// TwinCAT 3 PLC project ZeroTorque
// ProgramVersion: 3.1.4020.4
// libraries:
//   Tc2_MC2, * (Beckhoff Automation GmbH)
//   Tc2_Standard, * (Beckhoff Automation GmbH)
//   Tc2_System, * (Beckhoff Automation GmbH)
//   Tc3_Module, * (Beckhoff Automation GmbH)
// project tree:
//   GVLs/ GVL.TcGVL
//   / PlcTask.TcTTO
//   POUs/ KalmanFilter.TcPOU, MAIN.TcPOU
// real-time tasks:
//   TASK PlcTask: cycle T#10ms, priority 20, ADS port 350
// motion (NC):
//   TASK NC-Task 1 SAF: cycle T#2ms, priority 4, ADS port 501
//   TASK NC-Task 1 SVB: cycle T#10ms, priority 8, ADS port 511
//   AXIS Axis 1 (id 1)
//     Dynamic: AccelerationMaximum=150000, DecelerationMaximum=150000, Acceleration=5566, Deceleration=5566, Jerk=5566
//     Velo: SlowManual=50000, FastManual=150000, Maximum=150000
//     PositionAreaControl: Enable=false, RefSearch=false
//     TargetPosControl: Enable=false
//     OtherSettings: AllowMotionCmdToSlave=true
//     encoder EncType=19
//       EncPara: ScaleFactorNumerator=1, MaxCount=#xffffffff
//     drive DrvType=16
//       DrvPara: MaxCount=#xffffffff
//         Analog: VeloReferenz=150000
//         TimeComp: TaskDelayCycles=1
//     controller CtrType=1
//       CtrPara: PriorControlFactor=1
//         PosDiffControl: Enable=false
//         Observer: BandWidth=20
// I/O:
//   DEVICE Device 3 (EtherCAT), AmsNetId 172.18.138.230.4.1
//     Drive 1 (ZeroErr Driver) [ZeroErr Driver]
// variable links:
//   NC-Task 1 SAF/Axes/Axis 1 <-> Device 3 (EtherCAT)/Drive 1 (ZeroErr Driver)
//     Drive/Inputs/In/nDcOutputTime <-> InfoData/DcOutputShift
//     Drive/Inputs/In/nState1 <-> Transmit PDO mapping 0/Status word
//     Drive/Inputs/In/nState2 <-> Transmit PDO mapping 0/Status word @bit 8
//     Drive/Inputs/In/nState4 @bit 1 <-> WcState/InputToggle
//     Drive/Inputs/In/nState4 <-> WcState/WcState
//     Drive/Outputs/Out/nCtrl1 <-> Receive PDO mapping 0/Control word
//     Drive/Outputs/Out/nCtrl2 <-> Receive PDO mapping 0/Control word @bit 8
//     Drive/Outputs/Out/nDataOut1 <-> Receive PDO mapping 0/Target Position
//     Enc/Inputs/In/nDataIn1 <-> Transmit PDO mapping 0/Position actual value
//     Enc/Inputs/In/nDcInputTime <-> InfoData/DcInputShift
//     Enc/Inputs/In/nState4 @bit 1 <-> WcState/InputToggle
//     Enc/Inputs/In/nState4 <-> WcState/WcState
//   ZeroTorque/ZeroTorque Instance <-> Device 3 (EtherCAT)/Drive 1 (ZeroErr Driver)
//     PlcTask Inputs/GVL.ActTorque <-> Transmit PDO mapping 0/Current Actual Value
//     PlcTask Inputs/GVL.DualPosDiff <-> Transmit PDO mapping 0/Dual encoder difference value
//     PlcTask Inputs/GVL.actPosition <-> Transmit PDO mapping 0/Position actual value_1
//     PlcTask Inputs/GVL.actVelo <-> Transmit PDO mapping 0/Actual velocity
//     PlcTask Outputs/GVL.siOperationMode <-> Receive PDO mapping 0/Modes of operation
//     PlcTask Outputs/GVL.targetTor <-> Receive PDO mapping 0/Target Torque
//     PlcTask Outputs/GVL.targetVelo <-> Receive PDO mapping 0/Target Velocity
//     PlcTask Outputs/GVL.udiProAcc <-> Receive PDO mapping 0/Profile acceleration
//     PlcTask Outputs/GVL.udiProDec <-> Receive PDO mapping 0/Profile deceleration
//     PlcTask Outputs/GVL.udiProVelo <-> Receive PDO mapping 0/Profile velocity

CONFIGURATION ZeroTorque
    RESOURCE PLC ON TwinCAT3
        TASK PlcTask(INTERVAL := T#10ms, PRIORITY := 20);
        PROGRAM MAIN WITH PlcTask : MAIN;
    END_RESOURCE
END_CONFIGURATION

// ---- GVLs/GVL.TcGVL
{attribute 'qualified_only'}
VAR_GLOBAL
	(*--- Triansmit PDO ---*)
	DualPosDiff       AT%I*   :DINT;
	ActTorque         AT%I*   :INT;
	actVelo           AT%I*   :DINT;
	loadPos           AT%I*   :DINT;
	motorPos          AT%I*   :DINT;
	actPosition       AT%I*   :DINT;
	(*--- Receive PDO ---*)
	targetTor         AT%Q*   :INT;
	targetVelo        AT%Q*   :DINT;
	targetPos         AT%Q*   :DINT;
	uiCtrl            AT%Q*   :UINT;
	siOperationMode   AT%Q*   :SINT;
	udiProVelo        AT%Q*   :UDINT;
	udiProAcc         AT%Q*   :UDINT;
	udiProDec         AT%Q*   :UDINT;
	(*--- Control word bit ---*)
	arrCtrl           :ARRAY [0..15] OF BOOL;
	(*--- Status word bit ---*)
	arrStatus         :ARRAY [0..15] OF BOOL;
	(* process data*)
	dualPosFix         :DINT;
END_VAR

// ---- POUs/MAIN.TcPOU
PROGRAM MAIN
VAR
	iStep           :INT;
	timer1          :TON;
	referVelo       :DINT;
	sampleVelo      :DINT;//采样速度
	modAngle        :DINT;
	actAngle        :LREAL;
	rotation        :BOOL;//旋转方向
	rotationSingle  :INT;//旋转标志位
	runDirect       :INT;
	needChange      :BOOL;
	(*--- CSP ---*)
	axis1: AXIS_REF;
	power_do : BOOL;
	tarPosition : LREAL;
	oriPos      : DINT;//原始位置保存
	posSum      : DINT;
	posCount    :INT;
	ifPosModifyFinish : BOOL;
	tarVelocity : LREAL := 0;
	tarAcc      : LREAL := 50000;
	enable : BOOL:=TRUE;
	ifDone      :BOOL;
	ifGetTarPos :BOOL :=TRUE;
	K           :LREAL := 0.3;
	B           :LREAL := 0.5;
	BGain       :LREAL := 1;
	Bactual    	:LREAL;
	M           :LREAL := 0.5;
	iGain       :LREAL := 0.001;
	iLimit      :LREAL := 50000;
	veloLimit   :LREAL := 500;
	dualGain    :LREAL := 0.3;
	irDualPosFix   :LREAL;
	dualPosDiffPreFix :DINT;
	tarVelo :DINT := 0;
	posiDiff    :LREAL;
	sumPosDiff  :LREAL := 0;
	gainAcc : LREAL := 15;
	ifAction :BOOL := FALSE;
	(*--- For kalman filter ---*)
	filter1: KalmanFilter;
	filter2: KalmanFilter;
	irDualPos     : LREAL;//滤波后双编码器差值
	irActVelo: LREAL;
	(*--- Limit ---*)
	speedLimit: DINT   := 350;
	accMax:   UDINT  := 3000;
	accMin:   UDINT  := 200;
	(*--- Gain ---*)
	accGain   :LREAL   :=3;
	speedGain :DINT    :=50;
	dampGain  :LREAL   :=1.5;
	(*--- DeadZone ---*)
	deadZone       :LREAL   :=200;//驱动变速死区
	startDeadZone  :LREAL   :=150;//启动死区
	deadSpeedZone  :DINT    :=50;//速度归零死区
	(*--- Offset ---*)
	lowSpeedOffsetA   :LREAL :=872.783;//正低速偏置
	lowSpeedOffsetB   :LREAL :=860.311;//负低速偏置
	highSpeedOffsetA :LREAL :=772.06430;//正高速偏置
	highSpeedOffsetB :LREAL :=751.81464;//负高速偏置
	(*--- Offset Auto Modify---*)
	i                 : INT;
	offsetList        :ARRAY [0..99] OF LREAL;
	zeroCount         :INT   := 0;
	offsetSum         :LREAL := 0;
	offsetMean        :LREAL := 0;
	ifModifyFinish    :BOOL  := FALSE;

END_VAR

timer1(IN:= , PT:= T#0.5S, Q=> , ET=> );
CASE iStep OF
	0:
		GVL.uiCtrl:=6;//0x0006
		oriPos := GVL.actPosition;
		tarPosition := oriPos;
	1:
		GVL.udiProAcc:=1000;
		GVL.udiProDec:=1000;
		iStep:=2;
		timer1.IN:=TRUE;
	2:
		GVL.siOperationMode:=3;
		IF GVL.siOperationMode=3 THEN
			iStep:=10;//跳入使能
		END_IF
	10:	//使能
		//6
		IF GVL.uiCtrl = 0 THEN
			GVL.uiCtrl:=6;//0x002F
		END_IF
		IF timer1.Q THEN
			IF GVL.uiCtrl = 6 THEN
				GVL.uiCtrl:=47;//0x002F
				iStep:=15;//跳入运行
			END_IF
			timer1.IN:=FALSE;
		END_IF
	11://零力运行
		IF (GVL.actVelo > 45000) THEN
			GVL.dualPosFix:=GVL.DualPosDiff - (LREAL_TO_DINT(-(DINT_TO_LREAL(GVL.actVelo)*DINT_TO_LREAL(GVL.actVelo)*0.0000003816)+DINT_TO_LREAL(GVL.actVelo)*0.08359+highSpeedOffsetA));
		ELSIF (GVL.actVelo < -45000) THEN
			GVL.dualPosFix:=GVL.DualPosDiff - (LREAL_TO_DINT((DINT_TO_LREAL(GVL.actVelo)*DINT_TO_LREAL(GVL.actVelo)*0.0000003500)+DINT_TO_LREAL(GVL.actVelo)*0.07837+highSpeedOffsetB));
		ELSE
			GVL.dualPosFix:=GVL.DualPosDiff - (LREAL_TO_DINT(DINT_TO_LREAL(GVL.actVelo)*0.0624 + lowSpeedOffsetA));
		END_IF
		filter1(NewData:= GVL.dualPosFix, Q_cov:=, R_cov:= , OutData=> );
		irDualPos:=filter1.OutData;
		sampleVelo := GVL.actVelo/257;//重新标定参考速度
		
		(*--- 重新设置静态偏置---*)
		IF (ABS(sampleVelo)) < 5 AND ifModifyFinish = FALSE THEN
			offsetList[zeroCount] := irDualPos;
			zeroCount:=zeroCount + 1;
		ELSE
			zeroCount:=0;
		END_IF
		IF zeroCount >= 100 THEN
			offsetSum := 0;
			FOR i := 0 TO 99 BY +1 DO
				offsetSum := offsetSum + offsetList[i];
				offsetList[i] := 0;
			END_FOR;
			offsetMean := offsetSum / 100;
			zeroCount := 0;
			lowSpeedOffsetA := lowSpeedOffsetA + offsetMean;
			offsetSum := 0;
			ifModifyFinish:=TRUE;
		END_IF
		(*--- 完成设置静态偏置---*)
		IF runDirect = 0 AND ifModifyFinish = TRUE THEN//处于零位置稳态
			IF (irDualPos - startDeadZone) > 0 THEN
				runDirect := -1;
				ifModifyFinish := FALSE;
			ELSIF (irDualPos + startDeadZone) < 0  THEN
				runDirect := 1;
				ifModifyFinish := FALSE;
			END_IF
		ELSIF (irDualPos - deadZone) > 0 THEN
			runDirect := -1;
		ELSIF (irDualPos + deadZone) < 0 THEN
			runDirect := 1;
		ELSIF ABS(irDualPos) <100 THEN//当从动态进入稳态时
			runDirect := 0;
		END_IF
		(*--- 加速度和速度设定---*)
		IF runDirect <> 0 THEN
			GVL.udiProAcc:=LREAL_TO_UDINT(ABS(irDualPos)*accGain);
			GVL.udiProDec:=LREAL_TO_UDINT(ABS(irDualPos)*accGain);
			GVL.targetVelo:=sampleVelo+speedGain*runDirect;
		ELSE
			GVL.udiProAcc:=LREAL_TO_UDINT(DINT_TO_LREAL(ABS(sampleVelo))*dampGain);
			GVL.udiProDec:=LREAL_TO_UDINT(DINT_TO_LREAL(ABS(sampleVelo))*dampGain);
			GVL.targetVelo:=0;
		END_IF
		
		(*--- 限幅 ---*)
		IF GVL.targetVelo>speedLimit THEN
			GVL.targetVelo:=speedLimit;
		ELSIF GVL.targetVelo<-speedLimit THEN
			GVL.targetVelo:=-speedLimit;
		END_IF
		IF GVL.udiProAcc>accMax THEN
			GVL.udiProAcc:=accMax;
		END_IF
		IF GVL.udiProDec>accMax THEN
			GVL.udiProDec:=accMax;
		END_IF
		IF GVL.udiProAcc<accMin THEN
			GVL.udiProAcc:=accMin;
		END_IF
		IF GVL.udiProDec<accMin THEN
			GVL.udiProDec:=accMin;
		END_IF
	12://按角度变速正向运行
		//计算当前角度
		modAngle:= ABS(GVL.actPosition MOD 524288);
		actAngle:= (DINT_TO_LREAL(modAngle)/524288)*360;
		//控制关节变速运动
		GVL.targetVelo:=(ABS(LREAL_TO_DINT((actAngle-180)*1.5)))+30;
	13://按角度变速反向运行
		//计算当前角度
		modAngle:= ABS(GVL.actPosition MOD 524288);
		actAngle:= (DINT_TO_LREAL(modAngle)/524288)*360;
		//控制关节变速运动
		GVL.targetVelo:=-(ABS(LREAL_TO_DINT((actAngle-180)*1.5)))-30;
	14://按角度变速正反向运行
		//计算当前角度
		modAngle:= ABS(GVL.actPosition MOD 524288);
		actAngle:= (DINT_TO_LREAL(modAngle)/524288)*360;
		IF rotation = 0 THEN
			IF actAngle < 180 THEN
				IF rotationSingle = 2 THEN//切换模式
					rotation := 1;
					rotationSingle := 3;
					GVL.targetVelo:=0;
				ELSE
					IF actAngle <= 5 THEN
						rotationSingle := 1;
					END_IF
					GVL.targetVelo:=(ABS(LREAL_TO_DINT(actAngle*1.5)))+30;
				END_IF	
			ELSIF actAngle >= 180 THEN
				IF actAngle >= 355 AND rotationSingle = 1 THEN
					rotationSingle := 2;
				END_IF
				GVL.targetVelo:=(ABS(LREAL_TO_DINT((360-actAngle)*1.5)))+30;
			END_IF
		ELSE 
			IF actAngle < 180 THEN
				IF actAngle <= 5 AND rotationSingle = 4 THEN
					rotationSingle := 5;
				END_IF
				GVL.targetVelo:=-(ABS(LREAL_TO_DINT(actAngle*1.5)))-30;
			ELSIF actAngle >= 180 THEN
				IF rotationSingle = 5 THEN//切换模式
					rotation := 0;
					rotationSingle := 0;
					GVL.targetVelo:=0;
				ELSE
					IF actAngle >= 355 THEN
						rotationSingle := 4;
					END_IF
					GVL.targetVelo:=-(ABS(LREAL_TO_DINT((360-actAngle)*1.5)))-30;
				END_IF	
			END_IF
		END_IF
		//控制关节变速运动
		//GVL.targetVelo:=(ABS(LREAL_TO_DINT((actAngle-180)*1.5)))+30;
	15://二阶阻抗系统模拟
		(*--- 双编码器差值插补---*)
		IF GVL.actVelo > 45000 THEN
			GVL.dualPosFix:=GVL.DualPosDiff - (LREAL_TO_DINT(-(DINT_TO_LREAL(GVL.actVelo)*DINT_TO_LREAL(GVL.actVelo)*0.0000003665)+DINT_TO_LREAL(GVL.actVelo)*0.08170+highSpeedOffsetA));
		ELSIF GVL.actVelo < -45000 THEN
			GVL.dualPosFix:=GVL.DualPosDiff - (LREAL_TO_DINT((DINT_TO_LREAL(GVL.actVelo)*DINT_TO_LREAL(GVL.actVelo)*0.0000003247)+DINT_TO_LREAL(GVL.actVelo)*0.07503+highSpeedOffsetB));
		ELSIF GVL.actVelo > 0 THEN
			GVL.dualPosFix:=GVL.DualPosDiff - (LREAL_TO_DINT(DINT_TO_LREAL(GVL.actVelo)*0.06254 + lowSpeedOffsetA));
		ELSE
			GVL.dualPosFix:=GVL.DualPosDiff - (LREAL_TO_DINT(DINT_TO_LREAL(GVL.actVelo)*0.06284 + lowSpeedOffsetB));
		END_IF
		filter1(NewData:= GVL.dualPosFix, Q_cov:=, R_cov:= , OutData=> );
		irDualPos:=filter1.OutData;
		
		(*--- 重新设置静态偏置---*)
		IF (ABS(GVL.actVelo)) < 200 AND ifModifyFinish = FALSE THEN
			offsetList[zeroCount] := irDualPos;
			zeroCount:=zeroCount + 1;
		ELSE
			zeroCount:=0;
		END_IF
		IF zeroCount >= 100 THEN
			offsetSum := 0;
			FOR i := 0 TO 99 BY +1 DO
				offsetSum := offsetSum + offsetList[i];
				offsetList[i] := 0;
			END_FOR;
			offsetMean := offsetSum / 100;
			zeroCount := 0;
			lowSpeedOffsetA := lowSpeedOffsetA + offsetMean;
			lowSpeedOffsetB := lowSpeedOffsetB + offsetMean;
			offsetSum := 0;
			ifModifyFinish:=TRUE;
		END_IF
		
		(*--- 开始方向解算---*)
		IF runDirect = 0 AND ifModifyFinish = TRUE THEN//处于零位置稳态
			IF (irDualPos - startDeadZone) > 0 THEN
				runDirect := -1;
				ifAction := TRUE;
				ifModifyFinish := FALSE;
			ELSIF (irDualPos + startDeadZone) < 0  THEN
				runDirect := 1;
				ifAction := TRUE;
				ifModifyFinish := FALSE;
			END_IF
		ELSIF (irDualPos - deadZone) > 0 THEN
			runDirect := -1;
			ifAction := TRUE;
		ELSIF (irDualPos + deadZone) < 0 THEN
			runDirect := 1;
			ifAction := TRUE;
		ELSIF ABS(irDualPos) <100 THEN//当从动态进入稳态时
			runDirect := 0;
		END_IF
		
		(*--- 开始导纳控制解算---*)
		sampleVelo := GVL.actVelo/257;
		IF runDirect = 0 THEN//调整阻尼曲线
			Bactual := B + BGain * EXP(-ABS(oriPos - GVL.actPosition)/257);
		ELSE
			Bactual := B;
		END_IF
		//添加积分项并限幅
		posiDiff := (oriPos - DINT_TO_LREAL(GVL.actPosition))/257;
		sumPosDiff := sumPosDiff + posiDiff;
		IF sumPosDiff < -iLimit THEN
			sumPosDiff := -iLimit;
		ELSIF sumPosDiff > iLimit THEN
			sumPosDiff := iLimit;
		END_IF
		//调整外力曲线
		IF irDualPos < 500 AND irDualPos >= 0 THEN
			irDualPosFix := irDualPos * irDualPos /500;
		ELSIF irDualPos >= -500 AND irDualPos < 0 THEN
			irDualPosFix := -irDualPos * irDualPos /500;
		END_IF
		(*--- 运动状态判断---*)
		IF ifAction = TRUE AND runDirect = 0 AND ABS(sampleVelo) < 20 AND ABS(posiDiff) < 10 THEN
			ifAction := FALSE;
		END_IF
		(*--- 导纳控制---*)
		IF ifAction = TRUE THEN
			tarAcc := (-irDualPosFix * dualGain + iGain * sumPosDiff + K * posiDiff + Bactual*DINT_TO_LREAL(tarVelo - sampleVelo))/M;
			tarVelocity := tarVelocity + tarAcc * 0.01;
		ELSE//重置位置信息，去零漂
			tarAcc := 500;
			tarVelocity := 0;
			IF sampleVelo = 0 AND ifPosModifyFinish = FALSE THEN
				posCount := posCount + 1;
				posSum := posSum + GVL.actPosition;
				IF posCount = 100 THEN
					oriPos := posSum / 100;
					ifPosModifyFinish := TRUE;
				END_IF
			ELSE
				posCount := 0;
				posSum := 0;
			END_IF 
		END_IF
		
		IF tarVelocity > veloLimit THEN
			tarVelocity := veloLimit;
		ELSIF tarVelocity <= -veloLimit THEN
			tarVelocity := -veloLimit;
		END_IF
		
		tarAcc := tarAcc * gainAcc;
		(*--- 限幅 ---*)
		IF tarAcc>accMax THEN
			tarAcc:=accMax;
		ELSIF  tarAcc<=-LREAL_TO_DINT(accMax) THEN
			tarAcc:=-LREAL_TO_DINT(accMax);
		END_IF
		GVL.udiProAcc := LREAL_TO_UDINT(ABS(tarAcc));
		GVL.udiProDec := LREAL_TO_UDINT(ABS(tarAcc));
		
		(*--- 限幅 ---*)
		GVL.targetVelo := LREAL_TO_DINT(tarVelocity);
		IF GVL.targetVelo>speedLimit THEN
			GVL.targetVelo:=speedLimit;
		ELSIF GVL.targetVelo<-speedLimit THEN
			GVL.targetVelo:=-speedLimit;
		END_IF
	1000:
		GVL.targetVelo:=0;
		IF (ABS(gvl.actVelo)<1000) AND timer1.IN=FALSE THEN
			timer1.IN:=TRUE;
		END_IF
		IF timer1.Q THEN
			timer1.IN:=FALSE;
			iStep:=0;//停滞档
		END_IF
END_CASE

END_PROGRAM

// ---- POUs/KalmanFilter.TcPOU
FUNCTION_BLOCK KalmanFilter
VAR_INPUT
	NewData :LREAL;//预测值
	Q_cov   :LREAL:=2;//系统协方差，越大越相信预测
	R_cov   :LREAL:=100;//测量协方差，越大越相信旧测量值
END_VAR
VAR_OUTPUT
	OutData :LREAL;//真实值
END_VAR
VAR
	P_cov   :LREAL:=1;//k时刻先验协方差
	P1_cov  :LREAL;//k时刻后验协方差
	P2_cov  :LREAL;//k-1时刻后验协方差
	K       :LREAL;//卡尔曼增益
	Posterior:LREAL;//k时刻后验状态估计
	Posterior1:LREAL;//k-1时刻后验状态估计
	Priori    :LREAL;//k时刻先验状态估计
	a         :LREAL;
	b         :LREAL;
END_VAR

Priori:=Posterior1;
P_cov:=P2_cov+Q_cov;

K:=P_cov/(P_cov+R_cov);
Posterior:=Priori+K*(NewData-Priori);
P1_cov:=(1-K)*P_cov;

Posterior1:=Posterior;
P2_cov:=P1_cov;

OutData:=Posterior;

END_FUNCTION_BLOCK
